FUNCTION Handle_Movement : BOOL
VAR_INPUT
END_VAR
VAR
END_VAR

END_FUNCTION

(* stored: Version 1.1.0.1
   POU Handle_Movement: Id {b6b3d548-c2a6-4783-8489-7feef4129cea}, SpecialFunc None *)
